PROGRAM MAIN
VAR
END_VAR

END_PROGRAM

(* stored: Version 1.1.0.1
   POU MAIN: Id {63ec088f-5cb3-4756-bcca-d1bc8233f053} *)
